RoboDK station: kr10 targets.rdk

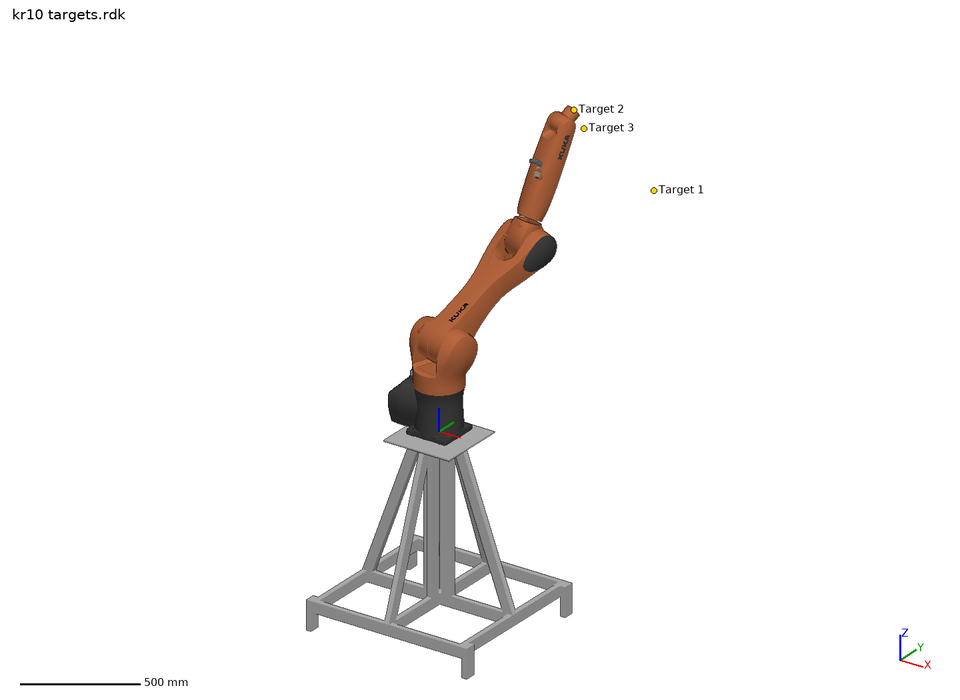
[picture v0: the station drawn from its stored meshes, robots at their saved joint values, targets as dots, program paths as lines]
Station kr10 targets. Poses are relative to the parent item; angles as X-Y-Z fixed-axis rotations.
  - frame KUKA KR 10 R1100 sixx Base at (0, 0, 0) mm
    - robot KUKA KR 10 R1100 sixx: 6 axes, payload 10 kg, reach 1101 mm, repeatability 0.03 mm, weight 54 kg
        modified DH rows (alpha deg, a mm, theta deg, d mm): 0, 0, 0, 400; -90, 25, 0, 0; 0, 560, -90, 0; -90, 35, 0, 515; 90, 0, 0, 0; -90, 0, 180, 80
        joint limits [-110, -190, -120, -185, -120, -350] to [110, 45, 156, 185, 120, 350]; home [0, -90, 90, 0, 0, 0]; saved at [-77.008, -34.206, -29.686, 7.149, 27.666, -344.615]
    - target Target 1 (Cartesian target) at (420.14, 952.98, 848.03) mm, rotated rx -24.18 ry 49.49 rz 42.34 deg; joints [-65.769, -7.254, -28.586, -97.037, 5.778, -247.881] of KUKA KR 10 R1100 sixx
    - target Target 2 (Cartesian target) at (172.58, 727.44, 1240.07) mm, rotated rx -24.18 ry 49.49 rz 42.34 deg; joints [-77.008, -34.206, -29.686, 7.149, 27.666, -344.615] of KUKA KR 10 R1100 sixx
    - target Target 3 (Cartesian target) at (139.16, 849.53, 1094.8) mm, rotated rx -24.18 ry 49.49 rz 42.34 deg; joints [-81.326, -20.269, -37.29, -161.578, -21.948, -172.866] of KUKA KR 10 R1100 sixx
    - target Target 4 (Cartesian target) at (172.58, 727.44, 1240.07) mm, rotated rx -24.18 ry 49.49 rz 42.34 deg; joints [-77.008, -34.206, -29.686, 7.149, 27.666, -344.615] of KUKA KR 10 R1100 sixx
  - object kuka base at (0, 0, 0) mm, size 812.8 x 762 x 857.2 mm, geometry from kuka base.stl
  - program Prog1 (4 instructions, listed below)

--- program Prog1 (robot KUKA KR 10 R1100 sixx) ---
  Set Ref.: KUKA KR 10 R1100 sixx Base
  Set speed (500.0 mm/s)
  MoveJ (Target 1)
  MoveL (Target 4)
